TEXTLIST TextList_Gaz
  0 = 'select' | FR: 'Sélectionner' | EN: 'Select'
  1 = 'ouvert' | FR: 'Ouverte' | EN: 'Opened'
  2 = 'fermé' | FR: 'Fermée' | EN: 'Closed'
  11 = 'ligne 1' | FR: 'Ligne de gaz 1' | EN: 'Gas line 1'
  12 = 'ligne 2' | FR: 'Ligne de gaz 2' | EN: 'Gas line 2'
  13 = 'ligne 3' | FR: 'Ligne de gaz 3' | EN: 'Gas line 3'
  14 = 'ligne 4' | FR: 'Ligne de gaz 4' | EN: 'Gas line 4'
  3 = 'debit' | FR: 'Débit (sccm)' | EN: 'Flow (sccm)'
  15 = 'Consigne pos' | FR: 'Consigne de position (%)' | EN: 'Position setpoint (%)'
  16 = 'Consigne pres' | FR: 'Consigne de pression (mbar)' | EN: 'Pressure setpoint (mbar)'
  17 = 'Press min' | FR: 'Pression min. (mbar)' | EN: 'Min. pressure (mbar)'
  18 = 'Press max' | FR: 'Pression max. (mbar)' | EN: 'Max. pressure (mbar)'
  19 = 'Temps stab' | FR: 'Temps de stab.' | EN: 'Stab. time'
   = ''
END_TEXTLIST

(* stored: Version 1.1.0.1, ProductVersion 3.1.4024.10
   TextList TextList_Gaz: Id {7d80d96e-8a3b-4910-981c-730ee4dc011a} *)
